// TIA Portal project "Box-Lifter Materialtransportsystem" (V16)
// Dieses Projekt simuliert ein automatisiertes Materialfördersystem mit einem Box-Lifter mithilfe von Siemens TIA Portal und einer S7-1200 SPS. Ziel ist die Realisierung eines kontinuierlichen Materialflusses mit Hilfe von Sensorik und Aktorik zur praxisnahen Anwendung sequentieller Steuerungen mit Zeitverzögerungen

(* hardware
DEVICE "S7-1200 station_1"  S7-1200 Station
   slot 0: "Rack_0"  S7-1200 Rack  Rack  V1.0
   slot 1: "PLC_1"  CPU 1214C AC/DC/Rly  6ES7 214-1BG31-0XB0  V3.0
*)

// ===== PLC "PLC_1"  CPU 1214C AC/DC/Rly =====

VAR_GLOBAL   // PLC tag table "Default tag table"
   "Stop_Taster" AT %I0.0 : Bool;   // Hält den Prozess an
   "Start_Taster" AT %I0.1 : Bool;   // Startet den Prozess
   "Sensor_box_vorhanden" AT %I0.2 : Bool;   // Sensor erkennt ankommende Box
   "Reed_Schalter" AT %I0.3 : Bool;   // Erkennt, ob Schieber wieder in Grundposition ist (homing)
   "Sensor_ladestation" AT %I0.4 : Bool;   // Sensor erkennt, dass die Box geladen ist
   "Sensor_Entladeposition" AT %I0.5 : Bool;   // Box am Ende Förderer 1
   "Motor_Förderkette" AT %Q0.1 : Bool;   // Förderbandmotor Ein/Aus
   "Schieber_Auswerfer" AT %Q0.2 : Bool;   // Schieber betätigen
   "Betriebsmodus" AT %M0.1 : Bool;   // Aktiver Zyklusstatus
END_VAR

// folder: System blocks/Program resources

DATA_BLOCK "T1"   // DB1
{ S7_Optimized_Access := 'TRUE' }
AUTHOR : Simatic
FAMILY : IEC
NAME : IEC_TMR
VERSION : 1.0
// stored: InstanceOfName IEC_TIMER
"IEC_TIMER"
BEGIN
END_DATA_BLOCK

DATA_BLOCK "T3"   // DB2
{ S7_Optimized_Access := 'TRUE' }
AUTHOR : Simatic
FAMILY : IEC
NAME : IEC_TMR
VERSION : 1.0
// stored: InstanceOfName IEC_TIMER
"IEC_TIMER"
BEGIN
END_DATA_BLOCK

DATA_BLOCK "IEC_Timer_0_DB"   // DB3
{ S7_Optimized_Access := 'TRUE' }
AUTHOR : Simatic
FAMILY : IEC
NAME : IEC_TMR
VERSION : 1.0
// stored: InstanceOfName IEC_TIMER
"IEC_TIMER"
BEGIN
END_DATA_BLOCK

DATA_BLOCK "T2"   // DB4
{ S7_Optimized_Access := 'TRUE' }
AUTHOR : Simatic
FAMILY : IEC
NAME : IEC_TMR
VERSION : 1.0
// stored: InstanceOfName IEC_TIMER
"IEC_TIMER"
BEGIN
END_DATA_BLOCK

// folder: (top level)

ORGANIZATION_BLOCK "Main"   // OB1, LAD, ProgramCycle
TITLE = "Main Program Sweep (Cycle)"
{ S7_Optimized_Access := 'TRUE' }
VERSION : 0.1
BEGIN

REGION Network 1: Förderbandmotor Ein/Aus
   // Start/Stopp-Logik (Motor aktiv)
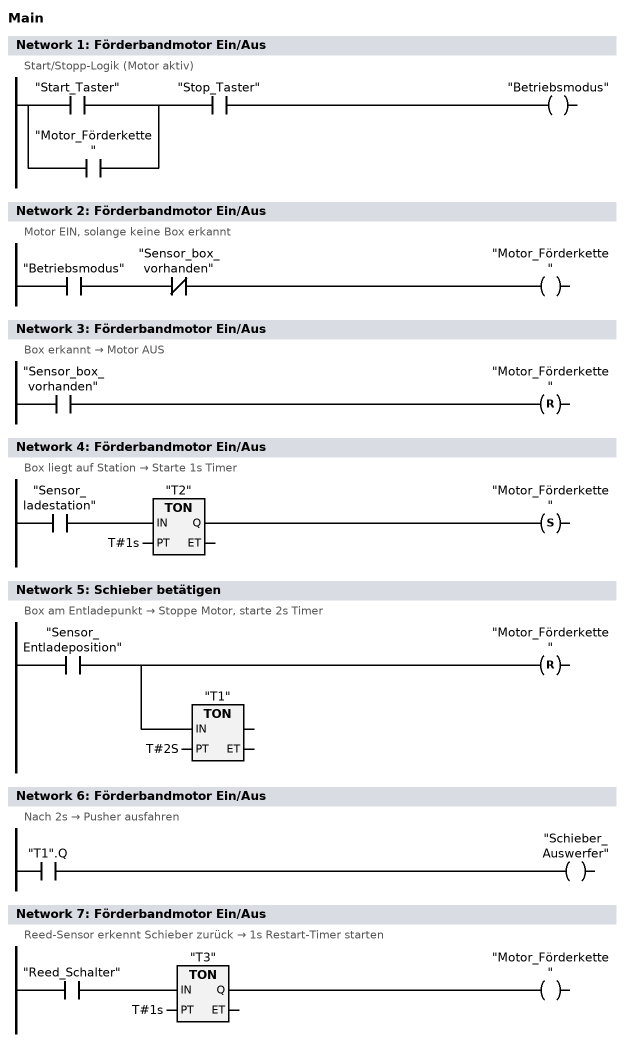
   RUNG wire#powerrail
      Contact( "Start_Taster" )
      wire#w1
      Contact( "Stop_Taster" )
      Coil( "Betriebsmodus" )
   END_RUNG
   RUNG wire#powerrail
      Contact( "Motor_Förderkette" )
   END_RUNG wire#w1
   // the same network as SCL:
   "Betriebsmodus" := ("Start_Taster" OR "Motor_Förderkette") AND "Stop_Taster";
END_REGION

REGION Network 2: Förderbandmotor Ein/Aus
   // Motor EIN, solange keine Box erkannt
   RUNG wire#powerrail
      Contact( "Betriebsmodus" )
      I_Contact( "Sensor_box_vorhanden" )
      Coil( "Motor_Förderkette" )
   END_RUNG
   // the same network as SCL:
   "Motor_Förderkette" := "Betriebsmodus" AND NOT "Sensor_box_vorhanden";
END_REGION

REGION Network 3: Förderbandmotor Ein/Aus
   // Box erkannt → Motor AUS
   RUNG wire#powerrail
      Contact( "Sensor_box_vorhanden" )
      R_Coil( "Motor_Förderkette" )
   END_RUNG
   // the same network as SCL:
   IF "Sensor_box_vorhanden" THEN "Motor_Förderkette" := FALSE; END_IF;
END_REGION

REGION Network 4: Förderbandmotor Ein/Aus
   // Box liegt auf Station → Starte 1s Timer
   "T2".TON(IN := "Sensor_ladestation", PT := T#1s);
   IF "T2".Q THEN "Motor_Förderkette" := TRUE; END_IF;
END_REGION

REGION Network 5: Schieber betätigen
   // Box am Entladepunkt → Stoppe Motor, starte 2s Timer
   IF "Sensor_Entladeposition" THEN "Motor_Förderkette" := FALSE; END_IF;
   "T1".TON(IN := "Sensor_Entladeposition", PT := T#2S);
END_REGION

REGION Network 6: Förderbandmotor Ein/Aus
   // Nach 2s → Pusher ausfahren
   RUNG wire#powerrail
      Contact( "T1".Q )
      Coil( "Schieber_Auswerfer" )
   END_RUNG
   // the same network as SCL:
   "Schieber_Auswerfer" := "T1".Q;
END_REGION

REGION Network 7: Förderbandmotor Ein/Aus
   // Reed-Sensor erkennt Schieber zurück → 1s Restart-Timer starten
   "T3".TON(IN := "Reed_Schalter", PT := T#1s);
   "Motor_Förderkette" := "T3".Q;
END_REGION
END_ORGANIZATION_BLOCK